{attribute 'GeneratedUsingTerminal: EPP3632-0001-0016'}
{attribute addProperty BoxType "EPP3632-0001-0016"}
{attribute addProperty Id "Ch1_ValueAT %I*INT2"}
{attribute addProperty CRC "2803750145"}
{attribute addProperty Size "2"}
TYPE Ch1_Sample_A71DD501 :
STRUCT
	{attribute addProperty Name "Ch1_Value"}
	Ch1_Value AT %I* : INT;
END_STRUCT
END_TYPE

(* stored: Version 1.2.0.0, ProductVersion 3.1.4024.9
   DUT Ch1_Sample_A71DD501: Id {ed99951a-46db-4533-8754-09192c6195f1} *)
